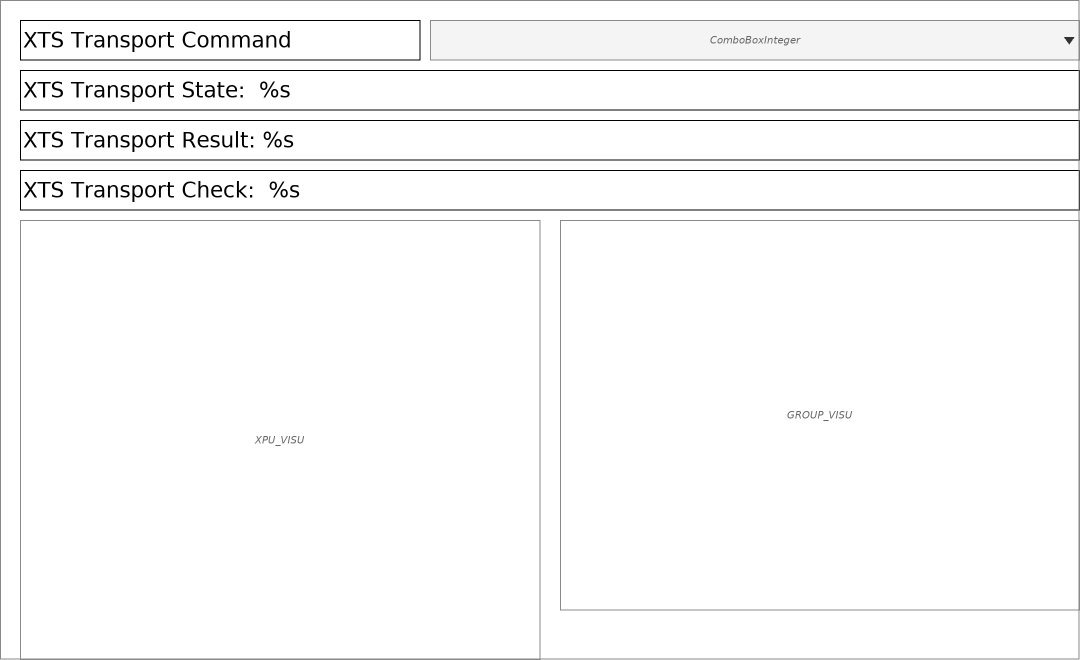
VISUALIZATION XTS_TRANSPORT  // 1080x660
    Rectangle (20,20 400x40), "XTS Transport Command"
    ComboBoxInteger (430,20 650x40), variable: GVL_XTS.XtsTransportCtrl.Cmd, text list: 'TL_E_CTRL_TRANSPORT'
    Rectangle (20,70 1060x40), "XTS Transport State: %s", text variable: MAIN.sTransportState
    Rectangle (20,120 1060x40), "XTS Transport Result: %s", text variable: MAIN.sTransportResult
    Rectangle (20,170 1060x40), "XTS Transport Check: %s", text variable: MAIN.sTransportCheck
    Frame (20,220 520x440)
        shows XPU_VISU(stXpuState := GVL_XTS.XtsTransportState.XpuState, stXpuInfo := GVL_XTS.XtsTransportState.XpuInfo, stXpuStrings := MAIN.stXpuStrings)
    Frame (560,220 520x390)
        shows GROUP_VISU(stGroupInfo := GVL_XTS.XtsTransportState.GroupInfo, sGroupState := MAIN.sCaGroupState)
END_VISUALIZATION

(* stored: Version 1.1.0.1
   Visu XTS_TRANSPORT: Id {34fe373c-43cd-4b86-9988-513bc9fa97ea} *)
